// TIA Portal project "交通红绿灯增强" (V20)

(* hardware
DEVICE "S7-1200 station_1"  S7-1200 Station
   slot 0: "Rack_0"  S7-1200 Rack  Rack  V1.0
   slot 1: "PLC_1"  CPU 1215C DC/DC/DC  6ES7 215-1AG40-0XB0  V4.6
   slot 3: "CB 1241 (RS485)"  CB 1241 (RS485)  6ES7 241-1CH30-1XB0  V1.0
*)

// ===== PLC "PLC_1"  CPU 1215C DC/DC/DC =====

VAR_GLOBAL   // PLC tag table "默认变量表"
   "Tag_1" AT %I0.0 : Bool;
END_VAR

DATA_BLOCK "数据块_1"   // DB1
{ S7_Optimized_Access := 'FALSE' }
VERSION : 0.1
// stored: InstanceOfName 块_1
"块_1"
BEGIN
END_DATA_BLOCK

FUNCTION_BLOCK "块_1"   // FB1, SCL
{ S7_Optimized_Access := 'FALSE' }
VERSION : 0.1
   VAR
      started : Bool;
      west_light : Struct
         green : Bool;
         yellow : Bool;
         red : Bool;
      END_STRUCT;
      south_light : Struct
         green : Bool;
         yellow : Bool;
         red : Bool;
      END_STRUCT;
      stage1 : Int;
      stage2 : Int;
      cnt : Int;
      IEC_Timer_0_Instance : TON_TIME;
      IEC_Timer_0_Instance_1 : TON_TIME;
      IEC_Timer_0_Instance_2 : TON_TIME;
   END_VAR
BEGIN
   IF "Tag_1" AND NOT #started THEN
       #started := 1;
       #stage1 := #stage2 := #cnt := 0;
       #west_light.green := #west_light.yellow := #west_light.red := #south_light.green := #south_light.yellow := #south_light.red := 0;
   END_IF;

   IF #west_light.green AND #south_light.green OR NOT #started THEN
       #west_light.green := #west_light.yellow := #west_light.red := #south_light.green := #south_light.yellow := #south_light.red := 0;
       #started := 0;
       #stage1 := #stage2 := #cnt := 0;
   END_IF;

   //start
   IF #stage1 = 0 AND #started AND #stage2 = 0 THEN
       #stage2 := 1;
       RESET_TIMER(#IEC_Timer_0_Instance);
   END_IF;
   //south red light
   IF #stage1 = 0 AND #stage2 = 1 THEN
       #south_light.red := 1;
       #west_light.green := 1;
       #IEC_Timer_0_Instance(IN := #stage2 = 1,
                             PT := t#20s);
       IF #IEC_Timer_0_Instance.Q THEN
           #stage2 += 1;
           #cnt := 0;
           RESET_TIMER(#IEC_Timer_0_Instance);
       END_IF;
   END_IF;

   IF #stage1 = 0 AND #stage2 = 2 THEN
       #IEC_Timer_0_Instance_1(IN := #stage2 = 2,
                               PT := t#0.5s);
       #IEC_Timer_0_Instance_2(IN := #IEC_Timer_0_Instance_1.Q,
                               PT := t#0.5s);
       #west_light.green := #IEC_Timer_0_Instance_1.Q;
       IF #IEC_Timer_0_Instance_2.Q THEN
           #cnt += 1;
           RESET_TIMER(#IEC_Timer_0_Instance_1);
           IF #cnt = 3 THEN
               #stage2 += 1;
               #cnt := 0;
               #west_light.green := 0;
           END_IF;
       END_IF;
   END_IF;

   IF #stage1 = 0 AND #stage2 = 3 THEN
       #west_light.yellow := 1;
       #IEC_Timer_0_Instance(IN := #stage2 = 3,
                             PT := t#2s);
       IF #IEC_Timer_0_Instance.Q THEN
           #stage2 := 1;
           #stage1 := 1;
           #south_light.red := 0;
           #west_light.yellow := 0;
           RESET_TIMER(#IEC_Timer_0_Instance);
       END_IF;
   END_IF;
   //west red light
   IF #stage1 = 1 AND #stage2 = 1 THEN
       #west_light.red := 1;
       #south_light.green := 1;
       #IEC_Timer_0_Instance(IN := #stage2 = 1,
                             PT := t#25s);
       IF #IEC_Timer_0_Instance.Q THEN
           #stage2 += 1;
           #cnt := 0;
           RESET_TIMER(#IEC_Timer_0_Instance);
       END_IF;
   END_IF;

   IF #stage1 = 1 AND #stage2 = 2 THEN
       #IEC_Timer_0_Instance_1(IN := #stage2 = 2,
                               PT := t#0.5s);
       #IEC_Timer_0_Instance_2(IN := #IEC_Timer_0_Instance_1.Q,
                               PT := t#0.5s);
       #south_light.green := #IEC_Timer_0_Instance_1.Q;
       IF #IEC_Timer_0_Instance_2.Q THEN
           #cnt += 1;
           RESET_TIMER(#IEC_Timer_0_Instance_1);
           IF #cnt = 3 THEN
               #stage2 += 1;
               #cnt := 0;
               #south_light.green := 0;
           END_IF;
       END_IF;
   END_IF;

   IF #stage1 = 1 AND #stage2 = 3 THEN
       #south_light.yellow := 1;
       #IEC_Timer_0_Instance(IN := #stage2 = 3,
                             PT := t#2s);
       IF #IEC_Timer_0_Instance.Q THEN
           #stage2 := 0;
           #stage1 := 0;
           #west_light.red := 0;
           #south_light.yellow := 0;
           RESET_TIMER(#IEC_Timer_0_Instance);
       END_IF;
   END_IF;
END_FUNCTION_BLOCK

ORGANIZATION_BLOCK "Main"   // OB1, LAD, ProgramCycle
TITLE = "Main Program Sweep (Cycle)"
{ S7_Optimized_Access := 'TRUE' }
VERSION : 0.1
   VAR_INPUT
      Initial_Call : Bool;   // Initial call of this OB
      Remanence : Bool;   // =True, if remanent data are available
   END_VAR
BEGIN

REGION Network 1
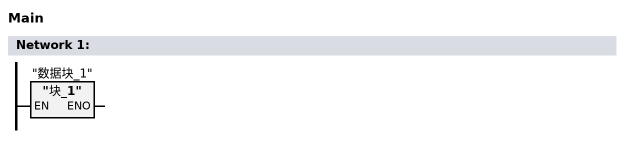
   RUNG wire#powerrail
      "数据块_1"()
   END_RUNG
   // the same network as SCL:
   "数据块_1"();   // "块_1"
END_REGION
END_ORGANIZATION_BLOCK